// TIA Portal V16 export
// export: Created 2022-11-14T17:35:42.8149215Z, ExportSetting WithDefaults, DisplayName Totally Integrated Automation Portal, DisplayVersion V16, DisplayName TIA Portal Version Control Interface, DisplayVersion V16, DisplayName TIA Portal Openness, DisplayVersion V16, DisplayName STEP 7 Professional, DisplayVersion V16, DisplayName STEP 7 Safety, DisplayVersion V16, DisplayName WinCC Advanced, DisplayVersion V16
DATA_BLOCK "DB23_AlarmProgram"   // DB23
{ S7_Optimized_Access := 'FALSE' }
AUTHOR : Robopac
VERSION : 0.0
// stored: AutoNumber false, IsOnlyStoredInLoadMemory false, IsWriteProtectedInAS false
   VAR RETAIN
      dbx0_0 : Bool := FALSE;   // Alarm 1: Pressure switch (Technoplat)
      dbx0_1 : Bool := FALSE;   // Alarm 2: Door open request (Technoplat)
      dbx0_2 : Bool := FALSE;   // Alarm 3: Emergency push button (Technoplat)
      dbx0_3 : Bool := FALSE;   // Alarm 4: Thermic alarm (Technoplat)
      dbx0_4 : Bool := FALSE;   // Alarm 5: Fault inverters (Technoplat)
      dbx0_5 : Bool := FALSE;   // Alarm 6: Motor start missing (Technoplat)
      dbx0_6 : Bool := FALSE;   // Alarm 7: Stop cycle by operator (Technoplat)
      dbx0_7 : Bool := FALSE;   // Alarm 8: Film ended or broken (Technoplat)
      dbx1_0 : Bool := FALSE;   // Alarm 9: Machine table not in phase (Technoplat)
      dbx1_1 : Bool := FALSE;   // Alarm 10: The spool carriage encoder is not running (Technoplat)
      dbx1_2 : Bool := FALSE;   // Alarm 11: Table encoder not working well
      dbx1_3 : Bool := FALSE;   // Alarm 12: Overspeed for table rotation (Technoplat)
      dbx1_4 : Bool := FALSE;   // Alarm 13: Phase table sensor lost (Technoplat)
      dbx1_5 : Bool := FALSE;   // Alarm 14: table deceleration not correct (Technoplat)
      dbx1_6 : Bool := FALSE;   // Alarm 15: Pressure plate not up (Pressure plate)
      dbx1_7 : Bool := FALSE;   // Alarm 16: Timeout for pressure plate upward/downward (Pressure plate)
      dbx2_0 : Bool := FALSE;   // Alarm 17: Pallet lifter not down (Lifter)
      dbx2_1 : Bool := FALSE;   // Alarm 18: Timeout for pallet lifter upward/downward (Lifter)
      dbx2_2 : Bool := FALSE;   // Alarm 19: Wrong data program for the pallet on the machine (Technoplat)
      dbx2_3 : Bool := FALSE;   // Alarm 20: Sysdata error (Technoplat)
      dbx2_4 : Bool := FALSE;   // Alarm 21: Spool carriage not down (Technoplat)
      dbx2_5 : Bool := FALSE;   // Alarm 22: Pressure plate positioning lost during rotation
      dbx2_6 : Bool := FALSE;   // Alarm 23:
      dbx2_7 : Bool := FALSE;   // Alarm 24: Emergency on infeed safety barrier (Barrier)
      dbx3_0 : Bool := FALSE;   // Alarm 25: Emergency on outfeed safety barrier (Barrier)
      dbx3_1 : Bool := FALSE;   // Alarm 26: Safety barrier excluded in automatic mode (Barrier)
      dbx3_2 : Bool := FALSE;   // Alarm 27: Timeout for rope unit open/close (Rope unit)
      dbx3_3 : Bool := FALSE;   // Alarm 28: Timeout for full rope unit open/close (Rope unit)
      dbx3_4 : Bool := FALSE;   // Alarm 29:
      dbx3_5 : Bool := FALSE;   // Alarm 30: Profinet communication error
      dbx3_6 : Bool := FALSE;   // Alarm 31: Modbus communication error
      dbx3_7 : Bool := FALSE;   // Alarm 32:
      dbx4_0 : Bool := FALSE;   // Alarm 33: Pallet positioning released during table rotation (Conveyor
      dbx4_1 : Bool := FALSE;   // Alarm 34: Pallet in transit in infeed (Conveyor)
      dbx4_2 : Bool := FALSE;   // Alarm 35: Pallet in transit in outfeed (Conveyor)
      dbx4_3 : Bool := FALSE;   // Alarm 36: Wrong pallet positioning (Conveyor)
      dbx4_4 : Bool := FALSE;   // Alarm 37: Infeed ring rotation control engaged (Conveyor)
      dbx4_5 : Bool := FALSE;   // Alarm 38: Outfeed ring rotation control engaged (Conveyor)
      dbx4_6 : Bool := FALSE;   // Alarm 39: Technoplat table not in load phase
      dbx4_7 : Bool := FALSE;   // Alarm 40: Technoplat table not in unload phase
      dbx5_0 : Bool := FALSE;   // Alarm 41: Contrast carriage not back
      dbx5_1 : Bool := FALSE;   // Alarm 42: Timeout contrast carriage forward/backward
      dbx5_2 : Bool := FALSE;   // Alarm 43: Clamp not closed (Clamp)
      dbx5_3 : Bool := FALSE;   // Alarm 44: Welder contrast not down (Clamp)
      dbx5_4 : Bool := FALSE;   // Alarm 45: Welder unit not down (Clamp)
      dbx5_5 : Bool := FALSE;   // Alarm 46: Clamp not down (Clamp)
      dbx5_6 : Bool := FALSE;   // Alarm 47: Welder contrast not up (Clamp)
      dbx5_7 : Bool := FALSE;   // Alarm 48: Timeout for clamp open/close (Clamp)
      dbx6_0 : Bool := FALSE;   // Alarm 49: Timeout for clamp upward/downward (Clamp)
      dbx6_1 : Bool := FALSE;   // Alarm 50: Timeout for welder contrast upward/downward (Clamp)
      dbx6_2 : Bool := FALSE;   // Alarm 51: Timeout for welder unit upward/downward (Clamp)
      dbx6_3 : Bool := FALSE;   // Alarm 52: Check the welder circuit (Clamp)
      dbx6_4 : Bool := FALSE;   // Alarm 53: Welder and cut unit not backward (Clamp)
      dbx6_5 : Bool := FALSE;   // Alarm 54: Timeout for welder and cut unit forward/backward (Clamp)
      dbx6_6 : Bool := FALSE;   // Alarm 55: Timeout for clamp carriage forward/backward (Clamp)
      dbx6_7 : Bool := FALSE;   // Alarm 56: Clamp carriage not backward (Clamp)
      dbx7_0 : Bool := FALSE;   // Alarm 57: Top carriage not up (Top)
      dbx7_1 : Bool := FALSE;   // Alarm 58: Top carriage not backward (Top)
      dbx7_2 : Bool := FALSE;   // Alarm 59: Top cutter not backward (Top)
      dbx7_3 : Bool := FALSE;   // Alarm 60: Clamp to pull top film not open (Top)
      dbx7_4 : Bool := FALSE;   // Alarm 61: Clamp to block top film not closed (Top)
      dbx7_5 : Bool := FALSE;   // Alarm 62: Top carriage not in position (Top)
      dbx7_6 : Bool := FALSE;   // Alarm 63: Top carriage not inside top film cut area (Top)
      dbx7_7 : Bool := FALSE;   // Alarm 64: Safety for top carriage position (Top)
      dbx8_0 : Bool := FALSE;   // Alarm 65: Timeout for top cutter (Top)
      dbx8_1 : Bool := FALSE;   // Alarm 66: Timeout for clamp to pull top film (Top)
      dbx8_2 : Bool := FALSE;   // Alarm 67: Timeout for clamp to block top film (Top)
      dbx8_3 : Bool := FALSE;   // Alarm 68: Top film ended or broken (Top)
      dbx8_4 : Bool := FALSE;   // Alarm 69: Infeed safety for top carriage up/down (Top)
      dbx8_5 : Bool := FALSE;   // Alarm 70: Outfeed safety for top carriage up/down (Top)
      dbx8_6 : Bool := FALSE;   // Alarm 71: Clamp to blok top film not open (Top)
      dbx8_7 : Bool := FALSE;   // Alarm 72: Top rele' brake broken (Top)
      dbx9_0 : Bool := FALSE;   // Alarm 73: Top not in position (Top inside signal)
      dbx9_1 : Bool := FALSE;   // Alarm 74: LIFTER POS.2 EXTRASTROKE UP
      dbx9_2 : Bool := FALSE;   // Alarm 75: LIFTER POS.2 FOOT SAFETY
      dbx9_3 : Bool := FALSE;   // Alarm 76: LIFTER POS.2 TIMEOUT CONVEYOR
      dbx9_4 : Bool := FALSE;   // Alarm 77: LIFTER POS.2 TIMEOUT UPSTROKE
      dbx9_5 : Bool := FALSE;   // Alarm 78: LIFTER POS.2 TIMEOUT DOWNSTROKE
      dbx9_6 : Bool := FALSE;   // Alarm 79: LABEL FAULT
      dbx9_7 : Bool := FALSE;   // Alarm 80: Label not in home position with table rotation
      dbx10_0 : Bool := FALSE;   // Alarm 81: Fire door not open during pallet transit
      dbx10_1 : Bool := FALSE;   // Alarm 82:
      dbx10_2 : Bool := FALSE;   // Alarm 83:
      dbx10_3 : Bool := FALSE;   // Alarm 84:
      dbx10_4 : Bool := FALSE;   // Alarm 85:
      dbx10_5 : Bool := FALSE;   // Alarm 86:
      dbx10_6 : Bool := FALSE;   // Alarm 87:
      dbx10_7 : Bool := FALSE;   // Alarm 88:
      dbx11_0 : Bool := FALSE;   // Alarm 89:
      dbx11_1 : Bool := FALSE;   // Alarm 90:
      dbx11_2 : Bool := FALSE;   // Alarm 91:
      dbx11_3 : Bool := FALSE;   // Alarm 92:
      dbx11_4 : Bool := FALSE;   // Alarm 93:
      dbx11_5 : Bool := FALSE;   // Alarm 94:
      dbx11_6 : Bool := FALSE;   // Alarm 95:
      dbx11_7 : Bool := FALSE;   // Alarm 96:
      dbx12_0 : Bool := FALSE;   // Alarm 97:
      dbx12_1 : Bool := FALSE;   // Alarm 98:
      dbx12_2 : Bool := FALSE;   // Alarm 99:
      dbx12_3 : Bool := FALSE;   // Alarm 100:
      dbx12_4 : Bool := FALSE;   // Alarm 101:
      dbx12_5 : Bool := FALSE;   // Alarm 102:
      dbx12_6 : Bool := FALSE;   // Alarm 103:
      dbx12_7 : Bool := FALSE;   // Alarm 104:
      dbx13_0 : Bool := FALSE;   // Alarm 105:
      dbx13_1 : Bool := FALSE;   // Alarm 106:
      dbx13_2 : Bool := FALSE;   // Alarm 107:
      dbx13_3 : Bool := FALSE;   // Alarm 108:
      dbx13_4 : Bool := FALSE;   // Alarm 109:
      dbx13_5 : Bool := FALSE;   // Alarm 110:
      dbx13_6 : Bool := FALSE;   // Alarm 111:
      dbx13_7 : Bool := FALSE;   // Alarm 112:
      dbx14_0 : Bool := FALSE;   // Alarm 113:
      dbx14_1 : Bool := FALSE;   // Alarm 114:
      dbx14_2 : Bool := FALSE;   // Alarm 115:
      dbx14_3 : Bool := FALSE;   // Alarm 116:
      dbx14_4 : Bool := FALSE;   // Alarm 117:
      dbx14_5 : Bool := FALSE;   // Alarm 118:
      dbx14_6 : Bool := FALSE;   // Alarm 119:
      dbx14_7 : Bool := FALSE;   // Alarm 120:
      dbx15_0 : Bool := FALSE;   // Alarm 121:
      dbx15_1 : Bool := FALSE;   // Alarm 122:
      dbx15_2 : Bool := FALSE;   // Alarm 123:
      dbx15_3 : Bool := FALSE;   // Alarm 124:
      dbx15_4 : Bool := FALSE;   // Alarm 125:
      dbx15_5 : Bool := FALSE;   // Alarm 126:
      dbx15_6 : Bool := FALSE;   // Alarm 127:
      dbx15_7 : Bool := FALSE;   // Alarm 128:
      dbx16_0 : Bool := FALSE;   // Alarm 129:
      dbx16_1 : Bool := FALSE;   // Alarm 130:
      dbx16_2 : Bool := FALSE;   // Alarm 131:
      dbx16_3 : Bool := FALSE;   // Alarm 132:
      dbx16_4 : Bool := FALSE;   // Alarm 133:
      dbx16_5 : Bool := FALSE;   // Alarm 134:
      dbx16_6 : Bool := FALSE;   // Alarm 135:
      dbx16_7 : Bool := FALSE;   // Alarm 136:
      dbx17_0 : Bool := FALSE;   // Alarm 137:
      dbx17_1 : Bool := FALSE;   // Alarm 138:
      dbx17_2 : Bool := FALSE;   // Alarm 139:
      dbx17_3 : Bool := FALSE;   // Alarm 140:
      dbx17_4 : Bool := FALSE;   // Alarm 141:
      dbx17_5 : Bool := FALSE;   // Alarm 142:
      dbx17_6 : Bool := FALSE;   // Alarm 143:
      dbx17_7 : Bool := FALSE;   // Alarm 144:
      dbx18_0 : Bool := FALSE;   // Alarm 145:
      dbx18_1 : Bool := FALSE;   // Alarm 146:
      dbx18_2 : Bool := FALSE;   // Alarm 147:
      dbx18_3 : Bool := FALSE;   // Alarm 148:
      dbx18_4 : Bool := FALSE;   // Alarm 149:
      dbx18_5 : Bool := FALSE;   // Alarm 150:
      dbx18_6 : Bool := FALSE;   // Alarm 151:
      dbx18_7 : Bool := FALSE;   // Alarm 152:
      dbx19_0 : Bool := FALSE;   // Alarm 153:
      dbx19_1 : Bool := FALSE;   // Alarm 154:
      dbx19_2 : Bool := FALSE;   // Alarm 155:
      dbx19_3 : Bool := FALSE;   // Alarm 156:
      dbx19_4 : Bool := FALSE;   // Alarm 157:
      dbx19_5 : Bool := FALSE;   // Alarm 158:
      dbx19_6 : Bool := FALSE;   // Alarm 159:
      dbx19_7 : Bool := FALSE;   // Alarm 160:
      dbx20_0 : Bool := FALSE;   // Alarm 161:
      dbx20_1 : Bool := FALSE;   // Alarm 162:
      dbx20_2 : Bool := FALSE;   // Alarm 163:
      dbx20_3 : Bool := FALSE;   // Alarm 164:
      dbx20_4 : Bool := FALSE;   // Alarm 165:
      dbx20_5 : Bool := FALSE;   // Alarm 166:
      dbx20_6 : Bool := FALSE;   // Alarm 167:
      dbx20_7 : Bool := FALSE;   // Alarm 168:
      dbx21_0 : Bool := FALSE;   // Alarm 169:
      dbx21_1 : Bool := FALSE;   // Alarm 170:
      dbx21_2 : Bool := FALSE;   // Alarm 171:
      dbx21_3 : Bool := FALSE;   // Alarm 172:
      dbx21_4 : Bool := FALSE;   // Alarm 173:
      dbx21_5 : Bool := FALSE;   // Alarm 174:
      dbx21_6 : Bool := FALSE;   // Alarm 175:
      dbx21_7 : Bool := FALSE;   // Alarm 176:
      dbx22_0 : Bool := FALSE;   // Alarm 177:
      dbx22_1 : Bool := FALSE;   // Alarm 178:
      dbx22_2 : Bool := FALSE;   // Alarm 179:
      dbx22_3 : Bool := FALSE;   // Alarm 180:
      dbx22_4 : Bool := FALSE;   // Alarm 181:
      dbx22_5 : Bool := FALSE;   // Alarm 182:
      dbx22_6 : Bool := FALSE;   // Alarm 183:
      dbx22_7 : Bool := FALSE;   // Alarm 184:
      dbx23_0 : Bool := FALSE;   // Alarm 185:
      dbx23_1 : Bool := FALSE;   // Alarm 186:
      dbx23_2 : Bool := FALSE;   // Alarm 187:
      dbx23_3 : Bool := FALSE;   // Alarm 188:
      dbx23_4 : Bool := FALSE;   // Alarm 189:
      dbx23_5 : Bool := FALSE;   // Alarm 190:
      dbx23_6 : Bool := FALSE;   // Alarm 191:
      dbx23_7 : Bool := FALSE;   // Alarm 192:
      dbx24_0 : Bool := FALSE;   // Alarm 193:
      dbx24_1 : Bool := FALSE;   // Alarm 194:
      dbx24_2 : Bool := FALSE;   // Alarm 195:
      dbx24_3 : Bool := FALSE;   // Alarm 196:
      dbx24_4 : Bool := FALSE;   // Alarm 197:
      dbx24_5 : Bool := FALSE;   // Alarm 198:
      dbx24_6 : Bool := FALSE;   // Alarm 199:
      dbx24_7 : Bool := FALSE;   // Alarm 200:
      dbx25_0 : Bool := FALSE;   // Alarm 201:
      dbx25_1 : Bool := FALSE;   // Alarm 202:
      dbx25_2 : Bool := FALSE;   // Alarm 203:
      dbx25_3 : Bool := FALSE;   // Alarm 204:
      dbx25_4 : Bool := FALSE;   // Alarm 205:
      dbx25_5 : Bool := FALSE;   // Alarm 206:
      dbx25_6 : Bool := FALSE;   // Alarm 207:
      dbx25_7 : Bool := FALSE;   // Alarm 208:
      dbx26_0 : Bool := FALSE;   // Warning 1: %10 Prestretch film on spool carriage (Technoplat)
      dbx26_1 : Bool := FALSE;   // Warning 2:
      dbx26_2 : Bool := FALSE;   // Warning 3: Request to reset encoder on spool carriage (Technoplat)
      dbx26_3 : Bool := FALSE;   // Warning 4:
      dbx26_4 : Bool := FALSE;   // Warning 5: Request to reset encoder on table rotation (Technoplat)
      dbx26_5 : Bool := FALSE;   // Warning 6:
      dbx26_6 : Bool := FALSE;   // Warning 7:
      dbx26_7 : Bool := FALSE;   // Warning 8: Fire door closing request
      dbx27_0 : Bool := FALSE;   // Warning 9: Timeout for door opening
      dbx27_1 : Bool := FALSE;   // Warning 10:
      dbx27_2 : Bool := FALSE;   // Warning 11:
      dbx27_3 : Bool := FALSE;   // Warning 12:
      dbx27_4 : Bool := FALSE;   // Warning 13:
      dbx27_5 : Bool := FALSE;   // Warning 14:
      dbx27_6 : Bool := FALSE;   // Warning 15:
      dbx27_7 : Bool := FALSE;   // Warning 16:
      dbx28_0 : Bool := FALSE;   // Warning 17:
      dbx28_1 : Bool := FALSE;   // Warning 18:
      dbx28_2 : Bool := FALSE;   // Warning 19:
      dbx28_3 : Bool := FALSE;   // Warning 20:
      dbx28_4 : Bool := FALSE;   // Warning 21:
      dbx28_5 : Bool := FALSE;   // Warning 22:
      dbx28_6 : Bool := FALSE;   // Warning 23:
      dbx28_7 : Bool := FALSE;   // Warning 24:
      dbx29_0 : Bool := FALSE;   // Warning 25:
      dbx29_1 : Bool := FALSE;   // Warning 26:
      dbx29_2 : Bool := FALSE;   // Warning 27:
      dbx29_3 : Bool := FALSE;   // Warning 28:
      dbx29_4 : Bool := FALSE;   // Warning 29:
      dbx29_5 : Bool := FALSE;   // Warning 30:
      dbx29_6 : Bool := FALSE;   // Warning 31:
      dbx29_7 : Bool := FALSE;   // Warning 32:
   END_VAR
BEGIN
END_DATA_BLOCK
